DATA_BLOCK "DB_OrinCommandStagingRaw"
{ S7_Optimized_Access := 'TRUE' }
VERSION : 0.1
NON_RETAIN
   VAR
      Registers : Array[0..63] of Word;
   END_VAR

BEGIN
END_DATA_BLOCK
